// TIA Portal V17 export
// export: Created 2024-01-30T08:49:13.5699506Z, ExportSetting WithDefaults, DisplayName Totally Integrated Automation Portal, DisplayVersion V17 Update 6, DisplayName TIA Portal Openness, DisplayVersion V17 Update 6, DisplayName TIA Portal Version Control Interface, DisplayVersion V17, DisplayName STEP 7 Professional, DisplayVersion V17 Update 6, DisplayName STEP 7 Safety, DisplayVersion V17 Update 6, DisplayName WinCC Advanced, DisplayVersion V17 Update 6
FUNCTION_BLOCK "LK_G5000"   // FB6, LAD
{ S7_Optimized_Access := 'TRUE' }
VERSION : 0.1
// stored: AutoNumber true, IsIECCheckEnabled false, IsRetainMemResEnabled false, MemoryReserve 100, SetENOAutomatically false, UDAEnableTagReadback false
BEGIN

REGION Network 1: Write / Read data in and from DB - CTRL_ BITS
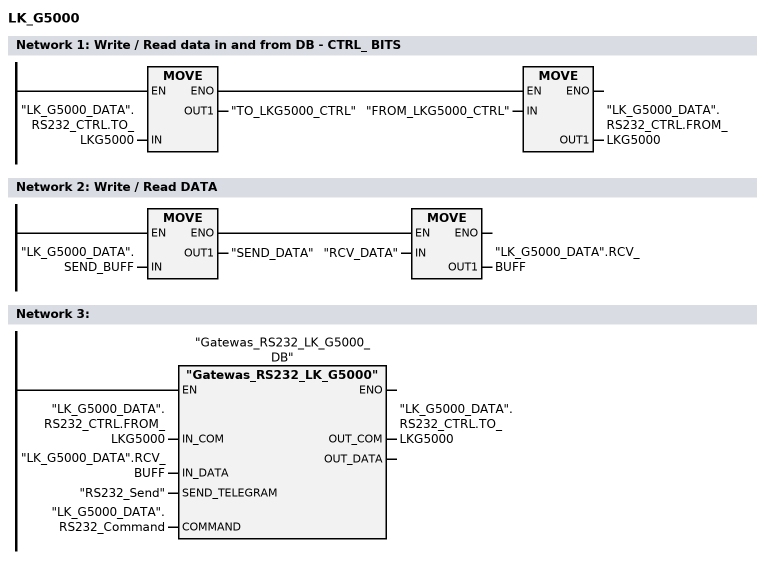
   RUNG wire#powerrail
      Move(in := "LK_G5000_DATA".RS232_CTRL.TO_LKG5000, out1 => "TO_LKG5000_CTRL")
      Move(in := "FROM_LKG5000_CTRL", out1 => "LK_G5000_DATA".RS232_CTRL.FROM_LKG5000)
   END_RUNG
   // the same network as SCL:
   "TO_LKG5000_CTRL" := "LK_G5000_DATA".RS232_CTRL.TO_LKG5000;
   "LK_G5000_DATA".RS232_CTRL.FROM_LKG5000 := "FROM_LKG5000_CTRL";
END_REGION

REGION Network 2: Write / Read DATA
   RUNG wire#powerrail
      Move(in := "LK_G5000_DATA".SEND_BUFF, out1 => "SEND_DATA")
      Move(in := "RCV_DATA", out1 => "LK_G5000_DATA".RCV_BUFF)
   END_RUNG
   // the same network as SCL:
   "SEND_DATA" := "LK_G5000_DATA".SEND_BUFF;
   "LK_G5000_DATA".RCV_BUFF := "RCV_DATA";
END_REGION

REGION Network 3
   RUNG wire#powerrail
      "Gatewas_RS232_LK_G5000_DB"(IN_COM := "LK_G5000_DATA".RS232_CTRL.FROM_LKG5000, IN_DATA := "LK_G5000_DATA".RCV_BUFF, SEND_TELEGRAM := "RS232_Send", COMMAND := "LK_G5000_DATA".RS232_Command, OUT_COM => "LK_G5000_DATA".RS232_CTRL.TO_LKG5000, OUT_DATA =>)
   END_RUNG
   // the same network as SCL:
   "Gatewas_RS232_LK_G5000_DB"(IN_COM := "LK_G5000_DATA".RS232_CTRL.FROM_LKG5000,   // "Gatewas_RS232_LK_G5000"
                           IN_DATA := "LK_G5000_DATA".RCV_BUFF,
                           SEND_TELEGRAM := "RS232_Send",
                           COMMAND := "LK_G5000_DATA".RS232_Command,
                           OUT_COM => "LK_G5000_DATA".RS232_CTRL.TO_LKG5000);
END_REGION
END_FUNCTION_BLOCK
